//{attribute 'qualified_only'}
VAR_GLOBAL


//	r_Accelerator_Setpoint	: REAL := 1E-12; (*unrealistic setpoint currently*)
    {attribute 'pytmc' := 'pv: TMO:FEE:VAC:OVRDON'}
    xSystemOverrideMode_FEE	: BOOL := FALSE; (* Global system override for the TMO FEE Vacuum System *)

    {attribute 'pytmc' := 'pv: TMO:NEH:VAC:OVRDON'}
    xSystemOverrideMode_TMO	: BOOL := FALSE; (* Global system override for the TMO hutch Vacuum System *)

    {attribute 'pytmc' := 'pv: TMO:NEH:TURBO:FAULT'}
    xTurboFault: BOOL := FALSE; (* True if any hutch turbo is not at speed or fault *)

    {attribute 'pytmc' := 'pv: TMO:NEH:VALVE:FAULT'}
    xBeamlineValveFault: BOOL := FALSE; (* True if any beamline valve is not open OK *)

        {attribute 'pytmc' := 'pv: TMO:NEH:ALL:GCC:ENABLE'}
    xGCC_Enable_SW: BOOL := FALSE; (* True if any hutch turbo is not at speed or fault *)

    {attribute 'pytmc' := 'pv: TMO:LAMP:PTM_NOK'}

    xLAMP_PTM_NOK AT%I*: BOOL := FALSE; (* True if any hutch turbo is not at speed or fault *)

    {attribute 'pytmc' := 'pv: TMO:VRC:DIFPRESS:BYPASS'}
    xBypassDiffPress_vrc1_vrc2 : BOOL;

    {attribute 'pytmc' := 'pv: TMO:FIM:HV_LOOP_PRESS'}
    iHV_LOOP_FIM_PRESSURE: REAL:= 8e-9;	//As Peter's request

    {attribute 'pytmc' := 'pv: TMO:FIM:HV_LOOP_ON'}
    {attribute 'TcLinkTo' := 'TIIB[K4S2_02_E20 (EL2004)]^Channel 4^Output'}
    iHV_LOOP_FIM_ON	AT %Q*: BOOL:= FALSE;

    {attribute 'pytmc' := 'pv: Pipe:replace:IP1'}
    xPipe_replace_IP1: BOOL := FALSE; (*tmo use piple to replace ip1 on  beamline*)

    {attribute 'pytmc' := 'pv: Psuedo:IP1:Gauge'}
    Psuedo_IP1_Gauge: ST_VG; //setup a psuedo gauge to select li2k4 instead of ip1 when pipe is in to replace ip1 08-21-25


END_VAR

(* stored: Version 1.1.0.1, ProductVersion 3.1.4024.12
   GVL GVL_Variables: Id {0b31be2f-6c9a-4798-a48f-4b64605f971e} *)
